FUNCTION_BLOCK FlushingManagerGSInstallation (* Basic Function Block Type *)
  (* Standard: 61499-2 *)
  (* Version 0.0, 8/23/2024, SESA713705, Schneider Electric, Template *)
  PACKAGE SE.Nereda;
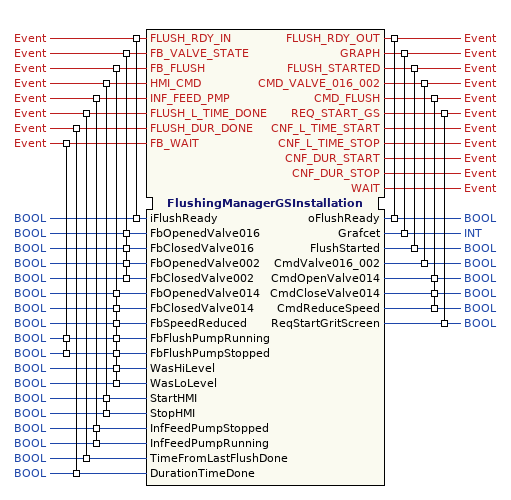
  EVENT_INPUT
    FLUSH_RDY_IN WITH iFlushReady;
    FB_VALVE_STATE WITH FbOpenedValve016, FbClosedValve016, FbOpenedValve002, FbClosedValve002;
    FB_FLUSH WITH FbOpenedValve014, FbClosedValve014, FbSpeedReduced, FbFlushPumpRunning, FbFlushPumpStopped, WasHiLevel, WasLoLevel;
    HMI_CMD WITH StartHMI, StopHMI;
    INF_FEED_PMP WITH InfFeedPumpStopped, InfFeedPumpRunning;
    FLUSH_L_TIME_DONE WITH TimeFromLastFlushDone;
    FLUSH_DUR_DONE WITH DurationTimeDone;
    FB_WAIT WITH FbFlushPumpRunning, FbFlushPumpStopped;
  END_EVENT
  EVENT_OUTPUT
    FLUSH_RDY_OUT WITH oFlushReady;
    GRAPH WITH Grafcet;
    FLUSH_STARTED WITH FlushStarted;
    CMD_VALVE_016_002 WITH CmdValve016_002;
    CMD_FLUSH WITH CmdOpenValve014, CmdCloseValve014, CmdReduceSpeed;
    REQ_START_GS WITH ReqStartGritScreen;
    CNF_L_TIME_START;
    CNF_L_TIME_STOP;
    CNF_DUR_START;
    CNF_DUR_STOP;
    WAIT;
  END_EVENT
  VAR_INPUT
    iFlushReady : BOOL;
    FbOpenedValve016 : BOOL;
    FbClosedValve016 : BOOL;
    FbOpenedValve002 : BOOL;
    FbClosedValve002 : BOOL;
    FbOpenedValve014 : BOOL;
    FbClosedValve014 : BOOL;
    FbSpeedReduced : BOOL;
    FbFlushPumpRunning : BOOL;
    FbFlushPumpStopped : BOOL;
    WasHiLevel : BOOL;
    WasLoLevel : BOOL;
    StartHMI : BOOL;
    StopHMI : BOOL;
    InfFeedPumpStopped : BOOL;
    InfFeedPumpRunning : BOOL;
    TimeFromLastFlushDone : BOOL;
    DurationTimeDone : BOOL;
  END_VAR
  VAR_OUTPUT
    oFlushReady : BOOL;
    Grafcet : INT;
    FlushStarted : BOOL;
    CmdValve016_002 : BOOL;
    CmdOpenValve014 : BOOL;
    CmdCloseValve014 : BOOL;
    CmdReduceSpeed : BOOL;
    ReqStartGritScreen : BOOL;
  END_VAR
  EC_STATES
    START; (* Initial State *)
    START_FLUSH : OpenValve016_002 -> CMD_VALVE_016_002, -> GRAPH;
    START_DUR : FlushStarted -> CNF_DUR_START, -> CNF_L_TIME_STOP, -> FLUSH_STARTED, -> GRAPH;
    STOP_FLUSH : CloseValve016_002 -> CMD_VALVE_016_002, -> GRAPH;
    FLUSH_OFF : FlushOFF -> CNF_L_TIME_START, -> CNF_DUR_STOP, -> REQ_START_GS, -> FLUSH_STARTED, -> FLUSH_RDY_OUT, -> GRAPH;
    ReduceSpeed2 : ReduceSpeed -> CMD_FLUSH, -> CNF_DUR_STOP, -> GRAPH;
    CloseValve14 : CloseValve014 -> CMD_FLUSH, -> GRAPH;
    InfFeedPumpRunning;
    FlushRdy : FlushRdy -> FLUSH_RDY_OUT, -> REQ_START_GS, -> GRAPH;
    ReduceSpeed1 : ReduceSpeed -> CMD_FLUSH, -> GRAPH;
    OpenValve014_1 : OpenValve014 -> CMD_FLUSH, -> GRAPH;
    CancelReduceSpeed : CancelReduceSpeed -> CMD_FLUSH, -> GRAPH;
    OpenValve014_2 : OpenValve014 -> CMD_FLUSH, -> GRAPH;
    CancelReduceSpeed1 : CancelReduceSpeed -> CMD_FLUSH, -> GRAPH;
    StopFlush;
    FlushingOFF : FlushingOFF -> FLUSH_RDY_OUT;
  END_STATES
  EC_TRANSITIONS
    InfFeedPumpRunning TO FlushRdy := iFlushReady AND TimeFromLastFlushDone AND InfFeedPumpStopped;
    START_FLUSH TO CloseValve14 := FbOpenedValve016 AND FbOpenedValve002;
    START_DUR TO ReduceSpeed2 := DurationTimeDone OR NOT iFlushReady;
    STOP_FLUSH TO CancelReduceSpeed1 := FbClosedValve016 AND FbClosedValve002;
    FLUSH_OFF TO START := 1;
    OpenValve014_2 TO STOP_FLUSH := FbOpenedValve014 OR FbFlushPumpStopped;
    CloseValve14 TO CancelReduceSpeed := FbClosedValve014;
    START TO InfFeedPumpRunning := INF_FEED_PMP AND InfFeedPumpRunning;
    START TO FlushRdy := HMI_CMD AND StartHMI AND NOT StopHMI;
    OpenValve014_1 TO ReduceSpeed1 := FbFlushPumpRunning;
    ReduceSpeed1 TO START_FLUSH := FbSpeedReduced;
    FlushRdy TO OpenValve014_1 := 1;
    CancelReduceSpeed TO START_DUR := NOT FbSpeedReduced;
    FlushingOFF TO OpenValve014_2 := WasHiLevel;
    CancelReduceSpeed1 TO FLUSH_OFF := NOT FbSpeedReduced OR FbFlushPumpStopped;
    OpenValve014_1 TO StopFlush := FB_WAIT AND FbFlushPumpStopped;
    ReduceSpeed1 TO StopFlush := FbFlushPumpStopped;
    START_FLUSH TO StopFlush := FbFlushPumpStopped;
    CloseValve14 TO StopFlush := FbFlushPumpStopped;
    CancelReduceSpeed TO StopFlush := FbFlushPumpStopped;
    START_DUR TO StopFlush := FbFlushPumpStopped;
    ReduceSpeed2 TO StopFlush := FbFlushPumpStopped;
    OpenValve014_2 TO StopFlush := FbFlushPumpStopped;
    StopFlush TO STOP_FLUSH := 1;
    InfFeedPumpRunning TO FlushRdy := HMI_CMD AND StartHMI AND NOT StopHMI;
    FlushingOFF TO STOP_FLUSH := WasLoLevel OR FbFlushPumpStopped;
    ReduceSpeed2 TO FlushingOFF := FbSpeedReduced;
  END_TRANSITIONS
  ALGORITHM OpenValve016_002 IN ST:
;
Grafcet := 4;
CmdValve016_002 := TRUE;
  END_ALGORITHM
  ALGORITHM FlushStarted IN ST:
;
Grafcet := 7;
FlushStarted := TRUE;
  END_ALGORITHM
  ALGORITHM CloseValve016_002 IN ST:
;
Grafcet := 10;
CmdValve016_002 := FALSE;
  END_ALGORITHM
  ALGORITHM FlushOFF IN ST:
;
Grafcet := 12;
CmdValve016_002 := FALSE;
FlushStarted := FALSE;
oFlushReady := FALSE;
ReqStartGritScreen := FALSE;
  END_ALGORITHM
  ALGORITHM OpenValve014 IN ST:
;
IF Grafcet = 1 THEN
	Grafcet := 2;
ELSIF Grafcet = 8 THEN
	Grafcet := 9;
END_IF;

CmdOpenValve014 := TRUE;
CmdCloseValve014 := FALSE;
  END_ALGORITHM
  ALGORITHM CancelReduceSpeed IN ST:
;
IF Grafcet = 5 THEN
	Grafcet := 6;
ELSIF Grafcet = 10 THEN
	Grafcet := 11;
END_IF;

CmdReduceSpeed := FALSE;
  END_ALGORITHM
  ALGORITHM FlushRdy IN ST:
;
Grafcet := 1;
IF StartHMI THEN
	oFlushReady := TRUE;
	ReqStartGritScreen := TRUE;
ELSE
	oFlushReady := iFlushReady;
END_IF;
  END_ALGORITHM
  ALGORITHM ReduceSpeed IN ST:
;
IF Grafcet = 2 THEN
	Grafcet := 3;
ELSIF Grafcet = 7 THEN
	Grafcet := 8;
END_IF;

CmdReduceSpeed := TRUE;
  END_ALGORITHM
  ALGORITHM CloseValve014 IN ST:
;
Grafcet := 5;
CmdOpenValve014 := FALSE;
CmdCloseValve014 := TRUE;
  END_ALGORITHM
  ALGORITHM FlushingOFF IN ST:
;
oFlushReady := FALSE;
  END_ALGORITHM
END_FUNCTION_BLOCK
